(* IEC 61131-3 sources: st2cpp/examples/tasks/src, 5 files *)

(* ---- counters.st ---- *)
(*
 * counters.st
 *
 * Global counters, incremented by the PROGRAM bodies. They exist so the example
 * can *show* how many times each program was invoked, which is the whole point
 * of the task configuration: the call counts are what tells you whether a task
 * really ran several programs, and whether a program shared between two tasks
 * was invoked once per task or only once in total.
 *
 * SimpleGVLs.hpp is what trace.cpp reads to print them.
*)

VAR_GLOBAL
    nMainCalls : DINT := 0;
    nControlCalls : DINT := 0;
    nReportCalls : DINT := 0;
END_VAR

(* ---- motor.st ---- *)
FUNCTION_BLOCK FB_Motor
VAR_INPUT
   nSetpoint : INT;
   bSteady   : BOOL;
END_VAR
VAR_OUTPUT
   nActual : INT;
END_VAR

IF bSteady THEN
   nActual := nSetpoint;
ELSE
   nActual := 0;
END_IF
END_FUNCTION_BLOCK

(* ---- report.st ---- *)
(*
 * report.st
 *
 * A third function block, so the example has three programs to distribute over
 * its tasks instead of two.
*)

FUNCTION_BLOCK FB_Report
VAR_INPUT
    bVerbose : BOOL;
END_VAR
VAR_OUTPUT
    nLines : INT;
END_VAR

IF bVerbose THEN
   nLines := 10;
ELSE
   nLines := 1;
END_IF
END_FUNCTION_BLOCK

(* ---- valve.st ---- *)
FUNCTION_BLOCK FB_Valve
VAR_INPUT
   bOpen : BOOL;
END_VAR
VAR_OUTPUT
   bIsOpen : BOOL;
END_VAR

bIsOpen := bOpen;
END_FUNCTION_BLOCK

(* ---- main.st ---- *)
(*
 * main.st
 *
 * The three PROGRAM POUs this example schedules. They are deliberately trivial
 * bodies: the interesting part is *which task calls which of them, and how
 * often*, which is what tasks.json declares.
*)

PROGRAM MAIN
VAR
    fbDrives : FB_Motor;
END_VAR

nMainCalls := nMainCalls + 1;
fbDrives(nSetpoint := 100);
END_PROGRAM

PROGRAM Control
VAR
    fbValve : FB_Valve;
END_VAR

nControlCalls := nControlCalls + 1;
fbValve(bOpen := TRUE);
END_PROGRAM

PROGRAM Report
VAR
    fbReport : FB_Report;
END_VAR

nReportCalls := nReportCalls + 1;
fbReport(bVerbose := FALSE);
END_PROGRAM
